PROGRAM MAIN
VAR
	Mercedes : coche;
	Bmw : coche;
	Audi: coche;
	
END_VAR

END_PROGRAM

(* stored: Version 1.1.0.1, ProductVersion 3.1.4024.12
   POU MAIN: Id {791988f4-6222-4a77-9850-9cca8d50763e}, SpecialFunc None *)
